// TIA Portal V20 export
// export: Created 2025-12-01T14:57:45.5461014Z, ExportSetting None, DisplayName Totally Integrated Automation Portal, DisplayVersion V20 Update 3, DisplayName TIA Portal Openness, DisplayVersion V20 Update 3, DisplayName TIA Portal Version Control Interface, DisplayVersion V20 Update 3, DisplayName STEP 7 Professional, DisplayVersion V20 Update 3, DisplayName STEP 7 Safety, DisplayVersion V20 Update 2, DisplayName WinCC Basic/Comfort/Advanced, DisplayVersion V20 Update 3, DisplayName WinCC Professional, DisplayVersion V20 Update 3, DisplayName WinCC Unified, DisplayVersion V20 Update 3
FUNCTION "FC893_Obtener_StringDelAtributo" : Void   // FC893, LAD
TITLE = "ObtenerStringAtributo" - Convertir a String un Doble Entero
{ S7_Optimized_Access := 'FALSE' }
AUTHOR : TRACKING
NAME : 20130301
VERSION : 3.0
// stored: AutoNumber false, SetENOAutomatically false
   VAR_INPUT
      DB_String : UInt;   // DB donde esta la String
      OffsetIni : UInt;   // Numero de byte de la String donde empieza
      Valor : UDInt;   // Valor a Convertir
   END_VAR
   VAR_OUTPUT
      OffsetFin : UInt;   // Numero de byte de la String donde acaba
   END_VAR
   VAR_TEMP
      PunteroDB : DWord;   // Puntero al DB de la String
      NumDB : Word;   // Num. del DB de la String
      ValorRestante : UDInt;   // Valor a convertir que va quedando
      OffsetActual : UInt;   // Numero de byte que estoy desplazando de la String
      Digito : UInt;   // Valor Convertiodo a Guardar en la String
      Temporal : UInt;
      TEMP_OffsetFin : UInt;
   END_VAR
BEGIN

NETWORK
TITLE = Inicializaciones
// Inicializar las Variables que se necesitan
      L     #Valor;  // Inicializo el Valor a Convertir
      T     #ValorRestante;

      L     #DB_String;
      T     #NumDB;

      L     #OffsetIni;  // Apunta al primer caracter el de Mayor peso
      T     #OffsetActual;
      T     #TEMP_OffsetFin;



NETWORK
TITLE = Conversion
// - Mirar si queda numero a convertir
// - Coger digito
// - Guardarlo en la String
// - Conseguir el Valor Restante
InicioBucle:NOP   0;

// -----------------------------------------------------------------------------------------------
// Coger el digito que necesitamos porner en la String - Menor peso

      L     #ValorRestante;
      L     10;
      MOD;  // Obtenemos el digito
      L     W#16#30;  // Y lo convertimos a Char
      +I;  // Sumar W#16#30
      T     #Digito;


// -----------------------------------------------------------------------------------------------
// Guardarlo en la String

      OPN   DB [#NumDB];

      L     #OffsetIni;  // Miro si es el Primer digito
      L     #TEMP_OffsetFin;
      ==I;
      JC    FinalDesplazar;  // Lo es

// Despalzar en la String para meter un nuevo digito

      L     #TEMP_OffsetFin;  // Inicializo al final
      T     #OffsetActual;  // Primer destino del desplazamiento
InicioDesPlazar:L     #OffsetActual;  // Recogo el dato del Byte Origen
      L     1;
      -I;
      SLD   3;
      T     #PunteroDB;
      L     DBB [#PunteroDB];
      T     #Temporal;

      L     #OffsetActual;  // Dejo el dato del Byte Destino
      SLD   3;
      T     #PunteroDB;
      L     #Temporal;
      T     DBB [#PunteroDB];

      L     #OffsetActual;  // Quito un digito para pasra el Siguiente
      L     1;
      -I;
      T     #OffsetActual;

      L     #OffsetActual;  // Se mira si estan todos desplazados
      L     #OffsetIni;
      ==I;
      JC    FinalDesplazar;  // Si estan todos
      JU    InicioDesPlazar;

// Guardo el ultimo digito guardado - Es el más significativo por ahora

FinalDesplazar:L     #OffsetIni;  // Guardo el digito convertido
      SLD   3;
      T     #PunteroDB;
      L     #Digito;
      T     DBB [#PunteroDB];

      L     #TEMP_OffsetFin;  // Incremento el Puntero Final de la String
      L     1;
      +I;
      T     #TEMP_OffsetFin;

// -----------------------------------------------------------------------------------------------
// Conseguimos el Valor Restante

      L     #ValorRestante;  // Dividimos en 10 para sacar el nuevo valor
      L     10;
      /D;
      T     #ValorRestante;

// -----------------------------------------------------------------------------------------------
// Mirar si queda nuero a convertir

      L     #ValorRestante;  // Validamos de que se trata de un numero
      L     0;  // No debe ser: Valor Restante < 0
      <=D;
      JC    Final;  // Se acabado el numero

      JU    InicioBucle;  // Vamos a ver si hay más digitos



NETWORK
TITLE = Final
// Final de la Funcion
Final:NOP   0;

      L     #TEMP_OffsetFin;  // - Devuelvo el Offset Temporal
      T     #OffsetFin;


END_FUNCTION
